PROGRAM Axis01_Auto
VAR
//System_Bit
	Always_ON	:	BOOL	:=TRUE	;//상시 ON 
	Always_OFF	:	BOOL	:=FALSE	;//상시 OFF
END_VAR

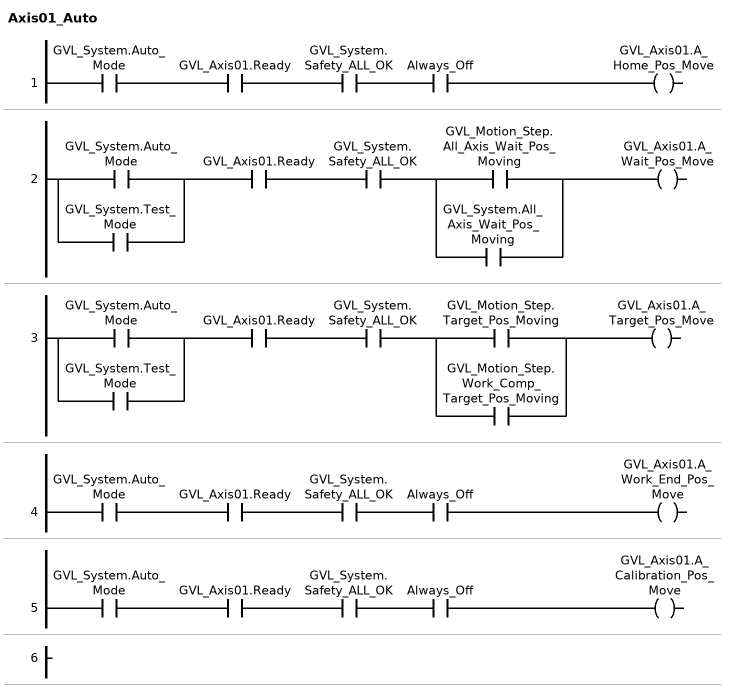
// NETWORK 1
GVL_Axis01.A_Home_Pos_Move := GVL_System.Auto_Mode AND GVL_Axis01.Ready AND GVL_System.Safety_ALL_OK AND Always_Off;

// NETWORK 2
GVL_Axis01.A_Wait_Pos_Move := (GVL_System.Auto_Mode OR GVL_System.Test_Mode) AND GVL_Axis01.Ready AND GVL_System.Safety_ALL_OK AND (GVL_Motion_Step.All_Axis_Wait_Pos_Moving OR GVL_System.All_Axis_Wait_Pos_Moving);

// NETWORK 3
GVL_Axis01.A_Target_Pos_Move := (GVL_System.Auto_Mode OR GVL_System.Test_Mode) AND GVL_Axis01.Ready AND GVL_System.Safety_ALL_OK AND (GVL_Motion_Step.Target_Pos_Moving OR GVL_Motion_Step.Work_Comp_Target_Pos_Moving);

// NETWORK 4
GVL_Axis01.A_Work_End_Pos_Move := GVL_System.Auto_Mode AND GVL_Axis01.Ready AND GVL_System.Safety_ALL_OK AND Always_Off;

// NETWORK 5
GVL_Axis01.A_Calibration_Pos_Move := GVL_System.Auto_Mode AND GVL_Axis01.Ready AND GVL_System.Safety_ALL_OK AND Always_Off;

// NETWORK 6

END_PROGRAM

(* stored: Version 1.1.0.1, ProductVersion 3.1.4024.16
   POU Axis01_Auto: Id {a556c58e-1b45-4a45-ad62-b9b9b34a80ae}, SpecialFunc None *)
